FUNCTION_BLOCK FB_EstacionVaciar_SFC

VAR_IN_OUT
	 TpoPreparacion: TIME;
     TpoMedidor: TIME;
END_VAR

VAR_INPUT
    // SFC-Flags
    SFCPause: BOOL;
    SFCReset: BOOL;
    
    // Indicadores de sincronizacion
    Ack: BOOL:= TRUE;
    Execute: BOOL;
	
	PlatoEmpujado: BOOL;
	PiezaRechazada: BOOL;
	PulsadorMarcha: BOOL;
	PiezaMedida: BOOL;
	Codificador: UINT;
    
END_VAR
VAR_OUTPUT
    // Indicadores de sincronizacion
    Done: BOOL;
    Ready: BOOL;
	EmpujaPlato : BOOL;
	RechazaPieza : BOOL;
	MedidorBaja: BOOL;
END_VAR
VAR
	Contador: INT;
    AuxiliarContador: INT;
	ListaAlturas : ARRAY[1..TAMANO_LISTA_PIEZAS] OF UINT;
END_VAR

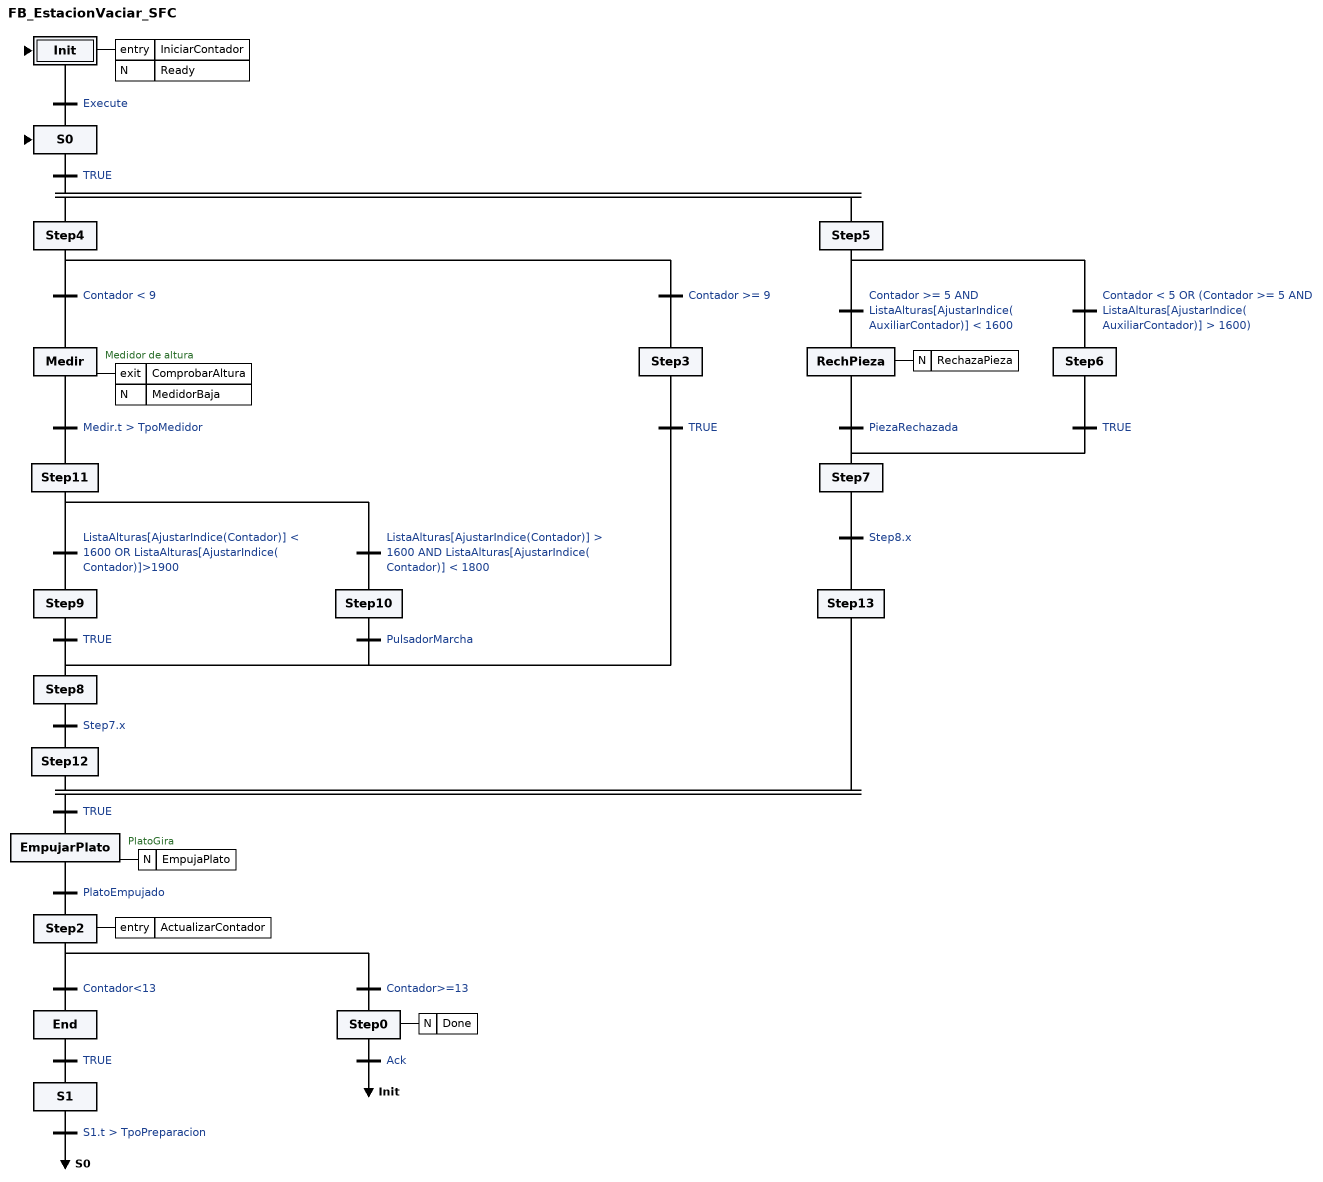
INITIAL_STEP Init:
    IniciarContador(P1);  // entry action
    Ready(N);
END_STEP
TRANSITION FROM Init TO S0
    := Execute;
END_TRANSITION
STEP S0:
END_STEP
TRANSITION FROM S0 TO (Step4, Step5)
    := TRUE;
END_TRANSITION
STEP Step4:
END_STEP
TRANSITION FROM Step4 TO Medir
    := Contador < 9;
END_TRANSITION
// Medidor de altura
STEP Medir:
    ComprobarAltura(P0);  // exit action
    MedidorBaja(N);
END_STEP
TRANSITION FROM Medir TO Step11
    := Medir.t > TpoMedidor;
END_TRANSITION
STEP Step11:
END_STEP
TRANSITION FROM Step11 TO Step9
    := ListaAlturas[AjustarIndice(Contador)] < 1600 OR ListaAlturas[AjustarIndice(Contador)]>1900;
END_TRANSITION
STEP Step9:
END_STEP
TRANSITION FROM Step9 TO Step8
    := TRUE;
END_TRANSITION
TRANSITION FROM Step11 TO Step10
    := ListaAlturas[AjustarIndice(Contador)] > 1600 AND ListaAlturas[AjustarIndice(Contador)] < 1800;
END_TRANSITION
STEP Step10:
END_STEP
TRANSITION FROM Step10 TO Step8
    := PulsadorMarcha;
END_TRANSITION
TRANSITION FROM Step4 TO Step3
    := Contador >= 9;
END_TRANSITION
STEP Step3:
END_STEP
TRANSITION FROM Step3 TO Step8
    := TRUE;
END_TRANSITION
STEP Step8:
END_STEP
TRANSITION FROM Step8 TO Step12
    := Step7.x;
END_TRANSITION
STEP Step12:
END_STEP
STEP Step5:
END_STEP
TRANSITION FROM Step5 TO RechPieza
    := Contador >= 5 AND ListaAlturas[AjustarIndice(AuxiliarContador)] < 1600;
END_TRANSITION
STEP RechPieza:
    RechazaPieza(N);
END_STEP
TRANSITION FROM RechPieza TO Step7
    := PiezaRechazada;
END_TRANSITION
TRANSITION FROM Step5 TO Step6
    := Contador < 5 OR (Contador >= 5 AND ListaAlturas[AjustarIndice(AuxiliarContador)] > 1600);
END_TRANSITION
STEP Step6:
END_STEP
TRANSITION FROM Step6 TO Step7
    := TRUE;
END_TRANSITION
STEP Step7:
END_STEP
TRANSITION FROM Step7 TO Step13
    := Step8.x;
END_TRANSITION
STEP Step13:
END_STEP
TRANSITION FROM (Step12, Step13) TO EmpujarPlato
    := TRUE;
END_TRANSITION
// PlatoGira
STEP EmpujarPlato:
    EmpujaPlato(N);
END_STEP
TRANSITION FROM EmpujarPlato TO Step2
    := PlatoEmpujado;
END_TRANSITION
STEP Step2:
    ActualizarContador(P1);  // entry action
END_STEP
TRANSITION FROM Step2 TO End
    := Contador<13;
END_TRANSITION
STEP End:
END_STEP
TRANSITION FROM End TO S1
    := TRUE;
END_TRANSITION
TRANSITION FROM Step2 TO Step0
    := Contador>=13;
END_TRANSITION
STEP Step0:
    Done(N);
END_STEP
TRANSITION FROM Step0 TO Init
    := Ack;
END_TRANSITION
STEP S1:
END_STEP
TRANSITION FROM S1 TO S0
    := S1.t > TpoPreparacion;
END_TRANSITION

ACTION ActualizarContador:
Contador := Contador + 1;
AuxiliarContador := Contador - 4;
END_ACTION

ACTION ComprobarAltura:
ListaAlturas[contador] := Codificador;
END_ACTION

ACTION IniciarContador:
Contador := 1;
END_ACTION

END_FUNCTION_BLOCK

(* stored: Version 1.1.0.1, ProductVersion 3.1.4024.12
   POU FB_EstacionVaciar_SFC: Id {d3fe0cf5-15ac-423d-b520-9cbba896411a}, SpecialFunc None
   Action ActualizarContador: Id {056e9552-6c71-4125-8986-c07f209b5840}
   Action ComprobarAltura: Id {f3628f25-4a12-409f-b5ea-84f76c392954}
   Action IniciarContador: Id {cffeacee-0dc1-4847-9499-e493e3acd434} *)
